FUNCTION_BLOCK FB_HeatPumpSystem EXTENDS FB_SystemContinous
VAR_INPUT
END_VAR
VAR_OUTPUT
END_VAR
VAR
	//Vitocal 350-G heat pump
	HeatPump : FB_HeatPump;
	
	//valve 146 and valve 246
	ST_SV146DefaultParameters : ST_DiscreteValveDefaultParameters := (bFeedbackSignal := FALSE);
	ST_SV246DefaultParameters : ST_DiscreteValveDefaultParameters := (bFeedbackSignal := FALSE);	
	SV146 : FB_DiscreteValve := (ST_DefaultParameters := ST_SV146DefaultParameters);
	SV246 : FB_DiscreteValve := (ST_DefaultParameters := ST_SV246DefaultParameters);	
	
	//internal variables
	bSetStatusOn_HeatPump : BOOL;
	bSetStatusOn_SV146 : BOOL;
	bSetStatusOn_SV246 : BOOL;
	
	bStartTimer : BOOL;
	Timer : TON;
END_VAR

MAIN();
//use timer because valve has no feedback signal (75 sec)
Timer(IN := bStartTimer,
	PT := T#75S);

//heat pump
HeatPump(bSetStatusOnAutomatic := bSetStatusOn_HeatPump,
	bAlgorithmPermission := bAlgorithmPermission);
HeatPump.SetState_BO();

//valves
SV146(bSetStatusOnAutomatic := bSetStatusOn_SV146,
		bAlgorithmPermission := bAlgorithmPermission);
SV146.SetState_BI_BO();
		
SV246(bSetStatusOnAutomatic := bSetStatusOn_SV246,
		bAlgorithmPermission := bAlgorithmPermission);
SV246.SetState_BI_BO();

METHOD PROTECTED  CheckError : BOOL
VAR_INPUT
END_VAR
VAR_OUTPUT
	bError : BOOL;
END_VAR
//empty method because system has no feedback signals
END_METHOD

METHOD PROTECTED  Operational : BOOL
VAR_INPUT
END_VAR
VAR_OUTPUT
	bSwitchToWorking : BOOL := FALSE;
END_VAR
bSetStatusOn_HeatPump := TRUE;
bSwitchToWorking := TRUE;
END_METHOD

METHOD PROTECTED  RampDown : BOOL
VAR_INPUT
END_VAR
VAR_OUTPUT
	bRampDownFinished : BOOL := FALSE;
END_VAR
bSetStatusOn_HeatPump := FALSE;
bSetStatusOn_SV146 := FALSE;
bSetStatusOn_SV246 := FALSE;
bStartTimer := TRUE;

IF Timer.Q THEN
	bRampDownFinished := TRUE;
	bStartTimer := FALSE;
END_IF
END_METHOD

METHOD PROTECTED  RampUp : BOOL
VAR_INPUT
END_VAR
VAR_OUTPUT
	bRampUpFinished : BOOL := FALSE;
END_VAR
bSetStatusOn_SV146 := TRUE;
bSetStatusOn_SV246 := TRUE;
bStartTimer := TRUE;

IF Timer.Q THEN
	bRampUpFinished := TRUE;
	bStartTimer := FALSE; //resets timer
END_IF
END_METHOD

METHOD PROTECTED   SetSetPointLimits : BOOL
VAR_INPUT
END_VAR
//heat pump has no continous setpoint (limits are not used) but must be implemented because of abstract method
aSetPointLimits[1] := 0;
aSetPointLimits[2] := 100;
END_METHOD

METHOD PROTECTED  Working : BOOL
VAR_INPUT
END_VAR
VAR_OUTPUT
	bSwitchToOperational : BOOL := FALSE;
END_VAR
//empty method because setpoint does not change during operation
END_METHOD

END_FUNCTION_BLOCK

(* stored: Version 1.1.0.1, ProductVersion 3.1.4024.9
   POU FB_HeatPumpSystem: Id {3b378086-0fcb-4a25-a8e9-ce86479d5246}, SpecialFunc None
   Method CheckError: Id {579f6d5c-ed17-4c3e-80e0-3652fdc92185}
   Method Operational: Id {e9fc807b-7078-4eae-9f16-4902d1f22c08}
   Method RampDown: Id {3e8b8560-8335-4c94-8f0e-af5b5bc8eb94}
   Method RampUp: Id {2dd804fd-9bc2-42b2-b115-7bf7a59d3046}
   Method SetSetPointLimits: Id {e4aed42f-62cc-4fb9-9793-37cfd06603ec}
   Method Working: Id {f8810774-f40a-40f9-b963-fb69028d850f} *)
